{attribute 'GeneratedUsingTerminal: ER1518-0002-0018'}
{attribute addProperty BoxType "ER1518-0002-0018"}
{attribute addProperty Id "ControlAT %Q*Control_0B2F8B702Set_counter_valueAT %Q*UDINT4"}
{attribute addProperty CRC "1426831071"}
{attribute addProperty Size "6"}
TYPE CNT_Output_Channel_550BB6DF :
STRUCT
	{attribute addProperty Name "Control"}
	Control AT %Q* : Control_0B2F8B70;
	{attribute addProperty Name "Set_counter_value"}
	Set_counter_value AT %Q* : UDINT;
END_STRUCT
END_TYPE

(* stored: Version 1.2.0.0, ProductVersion 3.1.4024.9
   DUT CNT_Output_Channel_550BB6DF: Id {09432bd9-3e0f-4cb4-9c50-747694bf837c} *)
